{attribute addProperty BoxType "EL5151-0021-0018"}
{attribute addProperty Id "ControlAT %Q*Control_2605F3141621Set_counter_valueAT %Q*UDINT32417Switch_on_threshold_valueAT %Q*UDINT32418Switch_off_threshold_valueAT %Q*UDINT32419"}
{attribute addProperty CRC "3762792797"}
{attribute addProperty SizeInBites "112"}
{attribute addProperty SizeInBytes "14"}
TYPE ENC_Control_E047A95D :
STRUCT
	{attribute addProperty Name "Control"}
	Control AT %Q* : Control_2605F314;
	{attribute addProperty Name "Set_counter_value"}
	Set_counter_value AT %Q* : UDINT;
	{attribute addProperty Name "Switch_on_threshold_value"}
	Switch_on_threshold_value AT %Q* : UDINT;
	{attribute addProperty Name "Switch_off_threshold_value"}
	Switch_off_threshold_value AT %Q* : UDINT;
END_STRUCT
END_TYPE

(* stored: Version 1.2.0.0, ProductVersion 3.1.4024.9
   DUT ENC_Control_E047A95D: Id {28b9f340-6773-4035-a1af-feb2508ca8be} *)
